INTERFACE I_Alarm EXTENDS I_Serializable

METHOD PUBLIC Accept
VAR_INPUT
	Visitor : I_AlarmVisitor;
END_VAR
END_METHOD

PROPERTY PUBLIC Active : BOOL
GET
END_GET
END_PROPERTY

PROPERTY PUBLIC Message : T_MaxString
GET
END_GET
END_PROPERTY

PROPERTY PUBLIC Reason : T_MaxString
GET
END_GET
END_PROPERTY

END_INTERFACE

(* stored: Version 1.1.0.1, ProductVersion 3.1.4024.12
   Itf I_Alarm: Id {86a2a33f-fdd7-41b8-9777-6da94dd2a119}
   Method Accept: Id {0a32d5aa-bebd-4bf3-b11b-e602cdcea0d5}
   Property Active: Id {84bfc066-f09c-42f2-8df7-e5e21a46d47a}
   Get Get: Id {70fa86e7-8487-49b4-a578-08410b0aa982}
   Property Message: Id {f47449c6-bd3b-48e4-a094-3b11b15515be}
   Get Get: Id {9d789d5f-bf78-4b41-ba80-c544ab35bf29}
   Property Reason: Id {87ad8f9d-b28e-4df2-af26-4da9a80b516e}
   Get Get: Id {d973eb1d-6672-42b5-bbc2-b792b7a04638} *)
